{attribute 'GeneratedUsingTerminal: EK1122-0000-0018'}
{attribute addProperty BoxType "EK1122-0000-0018"}
{attribute addProperty Id "Beckhoff_EK13xxsub_EK1100EK1100_1FC0878B2A_0001_EK1300_0000_0017EK1300_6BC01D146"}
{attribute addProperty CRC "819048514"}
{attribute addProperty Size "8"}
TYPE Beckhoff_EK13xxEK1122_30D1B042 EXTENDS EK1122_1FC0878B :
STRUCT
	{attribute addProperty Name "Beckhoff EK13xxsub EK1100"}
	{attribute addProperty PreviousPort "Beckhoff EK13xxEK1122 : D"}
	Beckhoff_EK13xxsub_EK1100 : EK1100_1FC0878B;
	{attribute addProperty Name "A_0001(EK1300-0000-0017)"}
	{attribute addProperty PreviousPort "Beckhoff EK13xxsub EK1100 : C"}
	A_0001_EK1300_0000_0017 : EK1300_6BC01D14;
END_STRUCT
END_TYPE

(* stored: Version 1.2.0.0, ProductVersion 3.1.4024.9
   DUT Beckhoff_EK13xxEK1122_30D1B042: Id {c19bf363-4aa8-4ebf-987f-e706c6ac473b} *)
